// Mitsubishi GX Works2 project: Cylinder   PLC: Q03UD

PROGRAM MAIN
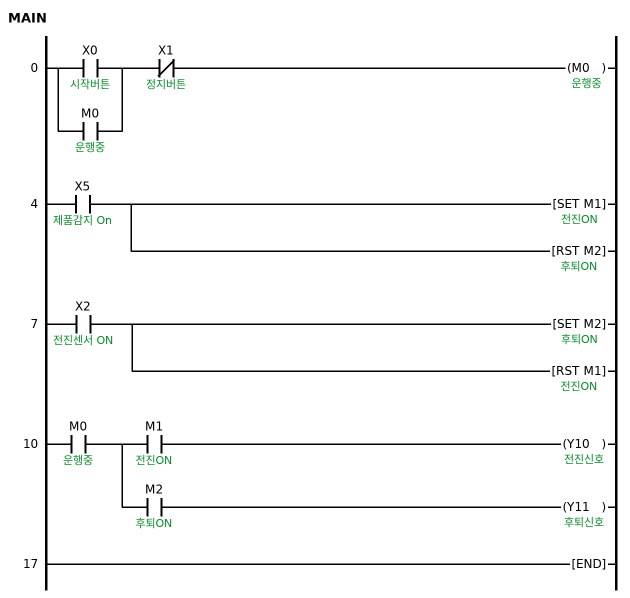
0     LD      X0  ; 시작버튼
      OR      M0  ; 운행중
      ANI     X1  ; 정지버튼
      OUT     M0  ; 운행중
4     LD      X5  ; 제품감지 On
      SET     M1  ; 전진ON
      RST     M2  ; 후퇴ON
7     LD      X2  ; 전진센서 ON
      SET     M2  ; 후퇴ON
      RST     M1  ; 전진ON
10    LD      M0  ; 운행중
      MPS
      AND     M1  ; 전진ON
      OUT     Y10  ; 전진신호
      MPP
      AND     M2  ; 후퇴ON
      OUT     Y11  ; 후퇴신호
17    END
END_PROGRAM

// device comments not shown above
X3  ; 후진센서 ON
